FUNCTION_BLOCK FB_VirtualControlBox IMPLEMENTS I_ControlBox
VAR_INPUT
END_VAR
VAR_OUTPUT
END_VAR
VAR
END_VAR

METHOD ModeSelector : BOOL
VAR_INPUT
	bOff	: BOOL;
	bManual	: BOOL;
	bAuto	: BOOL;
END_VAR
IF bOff THEN
	Work.eMode := E_Mode.Off;
END_IF

IF bManual THEN
	Work.eMode := E_Mode.Manual;
	Work.fJoystickY := VirtualControlBox.stVirtualInputs.fJoystickY;
END_IF

IF bAuto THEN
	Work.eMode := E_Mode.Auto;
END_IF
END_METHOD

END_FUNCTION_BLOCK

(* stored: Version 1.1.0.1, ProductVersion 3.1.4024.10
   POU FB_VirtualControlBox: Id {b5dbd877-8357-49f5-a98a-ac539e1b1d21}, SpecialFunc None
   Method ModeSelector: Id {e15f3617-ec38-4567-aa4b-7e33c463052d} *)
